FUNCTION_BLOCK Toggle IMPLEMENTS I_Toggle
VAR_INPUT
END_VAR
VAR_OUTPUT
END_VAR
VAR
	_ett: EntityStart;
		_component: Component(THIS^);
		_tag: Tag;
	_ettEnd: EntityEnd;
	
	_bValue: BOOL;
END_VAR

PROPERTY IsOn : BOOL
GET
IsOn := _bValue;
END_GET
END_PROPERTY

METHOD SwitchOff
_bValue := FALSE;
END_METHOD

METHOD SwitchOn
_bValue := TRUE;
END_METHOD

PROPERTY Tag : I_Tag
GET
Tag := _tag;
END_GET
END_PROPERTY

METHOD Toggle
_bValue := NOT _bValue;
END_METHOD

END_FUNCTION_BLOCK

(* stored: Version 1.1.0.1
   POU Toggle: Id {5b2ad2d0-5ba9-4b0b-92f7-57bc8abe23a7}, SpecialFunc None
   Property IsOn: Id {25abc126-dfb0-4e4e-ae2e-53fc96b45500}
   Get Get: Id {2da32b59-9795-477e-a06f-974942a5031e}
   Method SwitchOff: Id {4b025e55-3b74-4a40-b4ae-f89125dbf22b}
   Method SwitchOn: Id {2b989d0d-0fcd-444a-b99d-f52026e4cb83}
   Property Tag: Id {c3ebdb19-1735-4d55-883e-e69436a7b641}
   Get Get: Id {7ce2399c-e3d7-497b-a4bd-851028a71476}
   Method Toggle: Id {ad50040c-3f9a-4fe6-b7dc-d45beee4fd59} *)
